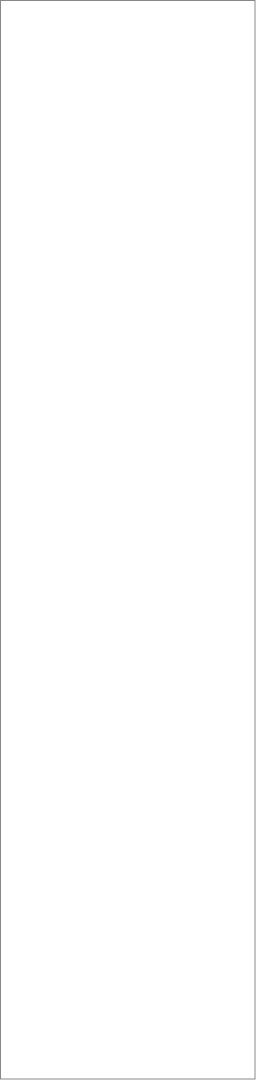
VISUALIZATION OtherList  // 256x1080
    Button (1413,1160 244x110), "ReM0"
        OnMouseDown: execute { G_HMI.iMainFrame  := 0; }
END_VISUALIZATION

(* stored: Version 1.1.0.1, ProductVersion 3.1.4024.12
   Visu OtherList: Id {c6646ba3-95c6-4885-9a92-385fe668c684} *)
